(* Logix 5000 project; controller Thurs_Lab2 vendor 1 type 14 code 156 rev 30.11; software revision 30.00; part 3 of 5 *)
(* tags used below, declared in another part *)
   Action_015 : SFC_ACTION;
   Action_016 : SFC_ACTION;
   Action_017 : SFC_ACTION;
   Action_018 : SFC_ACTION;
   Action_019 : SFC_ACTION;
   Action_020 : SFC_ACTION;
   Action_021 : SFC_ACTION;
   Action_022 : SFC_ACTION;
   Action_023 : SFC_ACTION;
   Action_024 : SFC_ACTION;
   Step_000 : SFC_STEP;
   Step_011 : SFC_STEP;
   Step_012 : SFC_STEP;
   Step_013 : SFC_STEP;
   Step_015 : SFC_STEP;
   Step_016 : SFC_STEP;
   Step_017 : SFC_STEP;
   Step_018 : SFC_STEP;
   Step_019 : SFC_STEP;
   Step_020 : SFC_STEP;
   Step_021 : SFC_STEP;
   Tran_000 : BOOL;
   AUTO : BOOL;
   BYPASS : BOOL;
   CONTINUE : BOOL;
   CYCLE_START : BOOL;
   CYCLE_STOP : BOOL;
   CYLINDERSTATUS : DINT;
   DEEP : COUNTER;
   DELAY_PE_INPUT_PSB : TIMER;
   DRILL2 : DRILL2;
   ESTOP_PRESSED : BOOL;
   EXTEND : TIMER;
   FAULT : BOOL;
   LOAD_ONE_SHOT_SCAN : BOOL;
   M_PL0 : BOOL;
   M_PL1 : BOOL;
   M_PL2 : BOOL;
   M_PL3 : BOOL;
   M_PL4 : BOOL;
   M_PL5 : BOOL;
   M_WHEEL_MOTOR : BOOL;
   Man_ONE_SHOT_SCAN : BOOL;
   Manual : BOOL;
   MARK_CYL1 : CYLINDER;
   MARK_ONE_SHOT_SCAN : BOOL;
   MASTER_RESET_COUNT1 : COUNTER;
   MASTER_RESET_COUNT2 : COUNTER;
   MASTER_RESET_COUNT3 : COUNTER;
   MASTER_RESET_COUNT4 : COUNTER;
   MASTER_RESET_COUNT5 : COUNTER;
   MASTER_RESET_COUNT6 : COUNTER;
   MASTER_RESET_COUNT7 : COUNTER;
   ONE_SHOT_PSB0 : BOOL;
   ONE_SHOT_PSB1 : BOOL;
   OP1_STOP : BOOL;
   OP2_ONE_SHOT_SCAN : BOOL;
   OP2_STEP : DINT;
   OP2_STOP : BOOL;
   OP3_ONE_SHOT_SCAN : BOOL;
   OP3_STOP : BOOL;
   OP4_ONE_SHOT_SCAN : BOOL;
   OP4_STOP : BOOL;
   OP5_STOP : BOOL;
   OP6_MARK : TIMER;
   OP6_STOP : BOOL;
   OP7_STOP : BOOL;
   OPERATION : DINT;
   OPERATION_DONE : DINT;
   OPERATION_OFF : DINT;
   OUTPUT : INT;
   PAUSE : BOOL;
   PB0 : BOOL;
   PB1 : BOOL;
   PB2 : BOOL;
   PB3 : BOOL;
   PB4 : BOOL;
   PB5 : BOOL;
   PV_CYL1_EXT_SIG : BOOL;
   PV_CYL1_RET_SIG : BOOL;
   PV_CYL2_EXT_SIG : BOOL;
   PV_FAULT_RESET : BOOL;
   PV_MAX_DEPTH : DINT;
   PV_MIN_DEPTH : DINT;
   PV_MOTOR_START : BOOL;
   PV_RESET : BOOL;
   RESET : BOOL;
   SAFETY_RELAY_OFF : BOOL;
   SEQ_EN : BOOL;
   SHALLOW : COUNTER;
   SORT_ONE_SHOT_SCAN : BOOL;
   START_SIGNAL : BOOL;
   STATE : DINT;
   STEP : DINT;
   TEST_ONE_SHOT_SCAN : BOOL;
   Timer : TIMER;
   TOO_DEEP : BOOL;
   TOO_SHALLOW : BOOL;
(* MainProgram, continued *)

ROUTINE MainRoutine   (* ladder *)
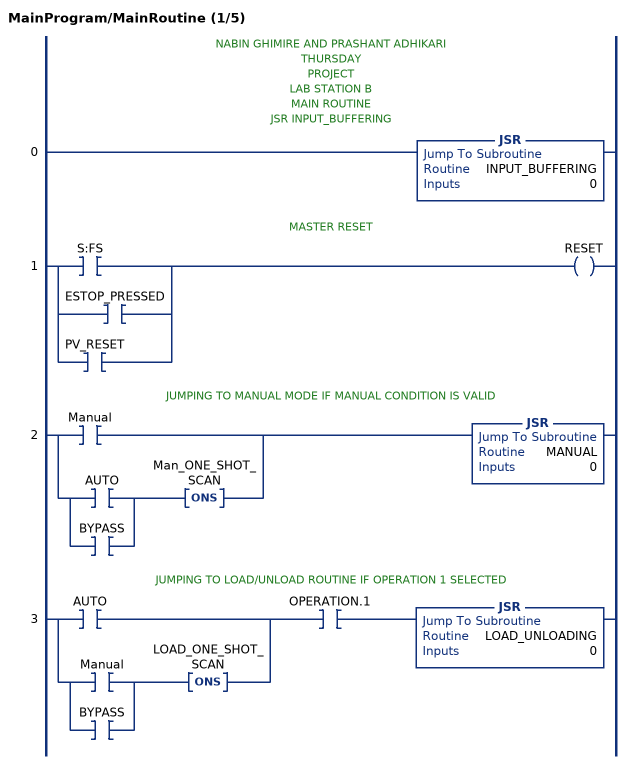
   // NABIN GHIMIRE AND PRASHANT ADHIKARI
   // THURSDAY
   // PROJECT
   // LAB STATION B
   // MAIN ROUTINE
   // JSR INPUT_BUFFERING
   0: JSR(INPUT_BUFFERING,0);
   // MASTER RESET
   1: [XIC(S:FS) ,XIC(ESTOP_PRESSED) ,XIC(PV_RESET) ]OTE(RESET);
   // JUMPING TO MANUAL MODE IF MANUAL CONDITION IS VALID
   2: [XIC(Manual) ,[XIC(AUTO) ,XIC(BYPASS) ] ONS(Man_ONE_SHOT_SCAN) ]JSR(MANUAL,0);
   // JUMPING TO LOAD/UNLOAD ROUTINE IF OPERATION 1 SELECTED
   3: [XIC(AUTO) ,[XIC(Manual) ,XIC(BYPASS) ] ONS(LOAD_ONE_SHOT_SCAN) ]XIC(OPERATION.1)JSR(LOAD_UNLOADING,0);
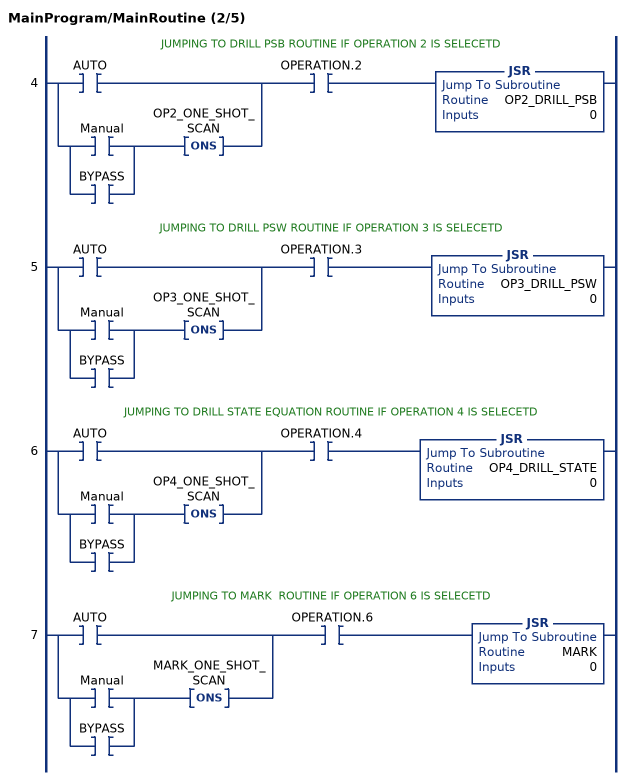
   // JUMPING TO DRILL PSB ROUTINE IF OPERATION 2 IS SELECETD
   4: [XIC(AUTO) ,[XIC(Manual) ,XIC(BYPASS) ] ONS(OP2_ONE_SHOT_SCAN) ]XIC(OPERATION.2)JSR(OP2_DRILL_PSB,0);
   // JUMPING TO DRILL PSW ROUTINE IF OPERATION 3 IS SELECETD
   5: [XIC(AUTO) ,[XIC(Manual) ,XIC(BYPASS) ] ONS(OP3_ONE_SHOT_SCAN) ]XIC(OPERATION.3)JSR(OP3_DRILL_PSW,0);
   // JUMPING TO DRILL STATE EQUATION ROUTINE IF OPERATION 4 IS SELECETD
   6: [XIC(AUTO) ,[XIC(Manual) ,XIC(BYPASS) ] ONS(OP4_ONE_SHOT_SCAN) ]XIC(OPERATION.4)JSR(OP4_DRILL_STATE,0);
   // JUMPING TO MARK  ROUTINE IF OPERATION 6 IS SELECETD
   7: [XIC(AUTO) ,[XIC(Manual) ,XIC(BYPASS) ] ONS(MARK_ONE_SHOT_SCAN) ]XIC(OPERATION.6)JSR(MARK,0);
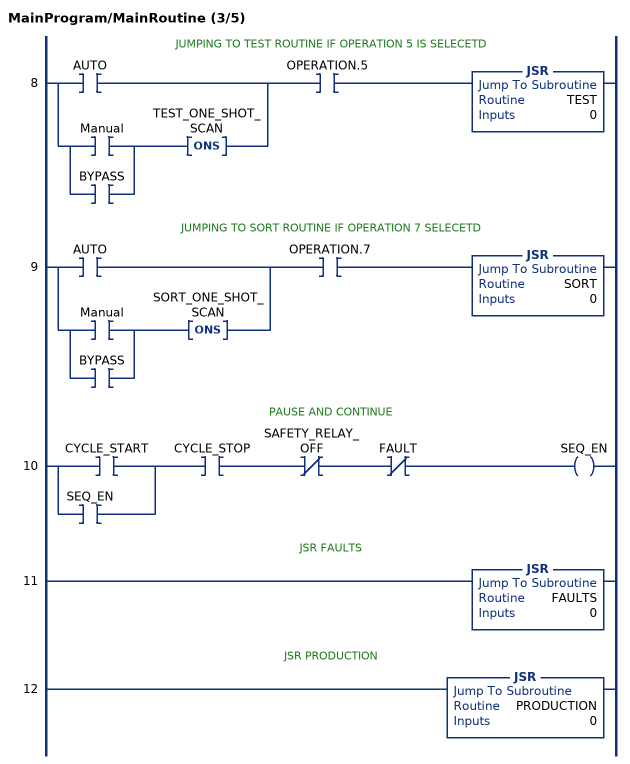
   // JUMPING TO TEST ROUTINE IF OPERATION 5 IS SELECETD
   8: [XIC(AUTO) ,[XIC(Manual) ,XIC(BYPASS) ] ONS(TEST_ONE_SHOT_SCAN) ]XIC(OPERATION.5)JSR(TEST,0);
   // JUMPING TO SORT ROUTINE IF OPERATION 7 SELECETD
   9: [XIC(AUTO) ,[XIC(Manual) ,XIC(BYPASS) ] ONS(SORT_ONE_SHOT_SCAN) ]XIC(OPERATION.7)JSR(SORT,0);
   // PAUSE AND CONTINUE
   10: [XIC(CYCLE_START) ,XIC(SEQ_EN) ]XIC(CYCLE_STOP)XIO(SAFETY_RELAY_OFF)XIO(FAULT)OTE(SEQ_EN);
   // JSR FAULTS
   11: JSR(FAULTS,0);
   // JSR PRODUCTION
   12: JSR(PRODUCTION,0);
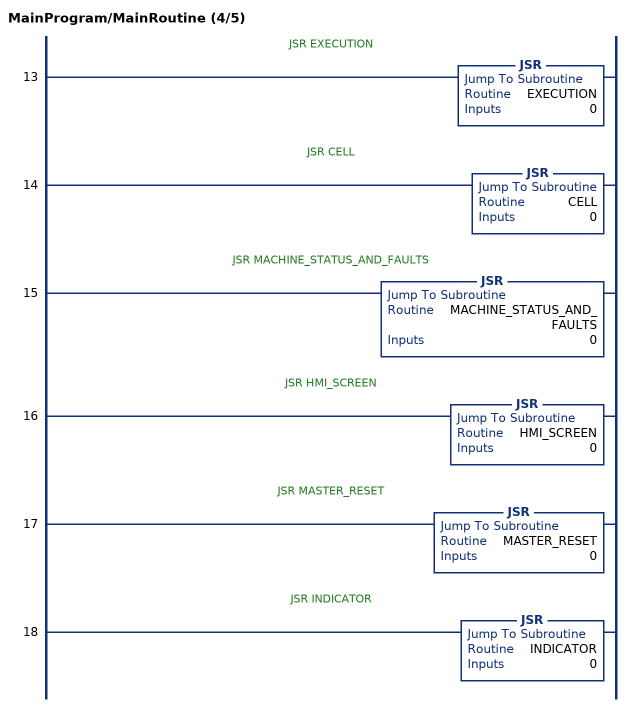
   // JSR EXECUTION
   13: JSR(EXECUTION,0);
   // JSR CELL
   14: JSR(CELL,0);
   // JSR MACHINE_STATUS_AND_FAULTS
   15: JSR(MACHINE_STATUS_AND_FAULTS,0);
   // JSR HMI_SCREEN
   16: JSR(HMI_SCREEN,0);
   // JSR MASTER_RESET
   17: JSR(MASTER_RESET,0);
   // JSR INDICATOR
   18: JSR(INDICATOR,0);
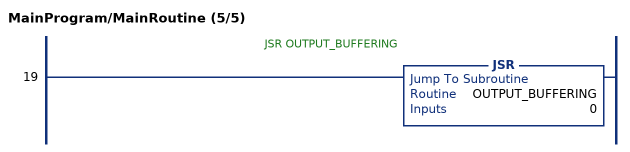
   // JSR OUTPUT_BUFFERING
   19: JSR(OUTPUT_BUFFERING,0);
END_ROUTINE

ROUTINE MANUAL   (* sequential function chart *)
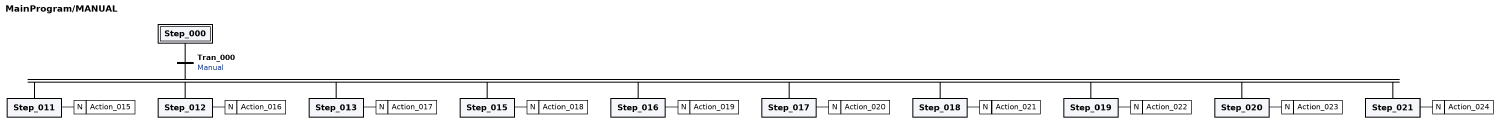
   // MANUAL ROUTINE USING SEQUENTIAL
   // FUNCTION CHART
   INITIAL_STEP Step_000:
   END_STEP
   TRANSITION Tran_000 FROM Step_000 TO (Step_012, Step_011, Step_013, Step_015, Step_016, Step_017, Step_018, Step_019, Step_020, Step_021)
      := Manual
         
         
   END_TRANSITION
   STEP Step_011:
      ACTION Action_015 (N):
         IF PB0 THEN
         	M_PL0:=1;
         ELSE
         	M_PL0:=0;
         END_IF;
         
         
      END_ACTION
   END_STEP
   STEP Step_012:
      ACTION Action_016 (N):
         IF PB1 THEN
         	M_PL1:=1;
         ELSE
         	M_PL1:=0;
         END_IF;
         
      END_ACTION
   END_STEP
   STEP Step_013:
      ACTION Action_017 (N):
         IF PB2 THEN
         	M_PL2:=1;
         ELSE
         	M_PL2:=0;
         END_IF;
         
      END_ACTION
   END_STEP
   STEP Step_015:
      ACTION Action_018 (N):
         IF PB3 THEN
         	M_PL3:=1;
         ELSE
         	M_PL3:=0;
         END_IF;
         
      END_ACTION
   END_STEP
   STEP Step_016:
      ACTION Action_019 (N):
         IF PB4 THEN
         	M_PL4:=1;
         ELSE
         	M_PL4:=0;
         END_IF;
         
      END_ACTION
   END_STEP
   STEP Step_017:
      ACTION Action_020 (N):
         IF PB5 THEN
         	M_PL5:=1;
         ELSE
         	M_PL5:=0;
         END_IF;
         
      END_ACTION
   END_STEP
   STEP Step_018:
      ACTION Action_021 (N):
         IF PV_MOTOR_START THEN
         	M_WHEEL_MOTOR:=1;
         ELSE
         	M_WHEEL_MOTOR:=0;
         END_IF;
         
      END_ACTION
   END_STEP
   STEP Step_019:
      ACTION Action_022 (N):
         IF PV_CYL2_EXT_SIG THEN
         	DRILL2.CYL2.EXT_SIG:=1;
         ELSE
         	DRILL2.CYL2.EXT_SIG:=0;
         END_IF;
         
      END_ACTION
   END_STEP
   STEP Step_020:
      ACTION Action_023 (N):
         IF PV_CYL1_RET_SIG THEN
         	DRILL2.CYL1.MAN_RET_SIG:=1;
         ELSE
         	DRILL2.CYL1.MAN_RET_SIG:=0;
         END_IF;
         
      END_ACTION
   END_STEP
   STEP Step_021:
      ACTION Action_024 (N):
         IF PV_CYL1_EXT_SIG THEN
         	DRILL2.CYL1.MAN_EXT_SIG:=1;
         ELSE
         	DRILL2.CYL1.MAN_EXT_SIG:=0;
         END_IF;
         
      END_ACTION
   END_STEP
END_ROUTINE

ROUTINE MARK   (* ladder *)
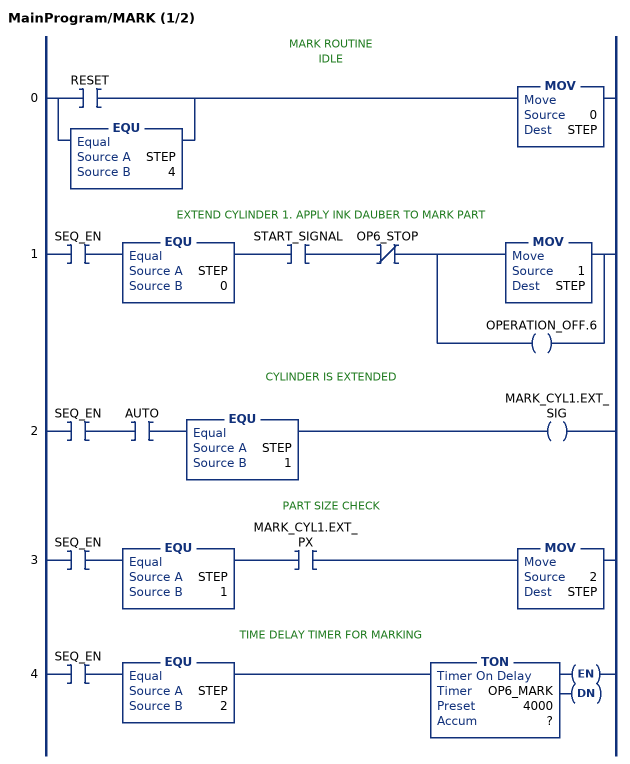
   // MARK ROUTINE
   // IDLE
   0: [XIC(RESET) ,EQU(STEP,4) ]MOV(0,STEP);
   // EXTEND CYLINDER 1. APPLY INK DAUBER TO MARK PART
   1: XIC(SEQ_EN)EQU(STEP,0)XIC(START_SIGNAL)XIO(OP6_STOP)[MOV(1,STEP) ,OTE(OPERATION_OFF.6) ];
   // CYLINDER IS EXTENDED
   2: XIC(SEQ_EN)XIC(AUTO)EQU(STEP,1)OTE(MARK_CYL1.EXT_SIG);
   // PART SIZE CHECK
   3: XIC(SEQ_EN)EQU(STEP,1)XIC(MARK_CYL1.EXT_PX)MOV(2,STEP);
   // TIME DELAY TIMER FOR MARKING
   4: XIC(SEQ_EN)EQU(STEP,2)TON(OP6_MARK,?,?);
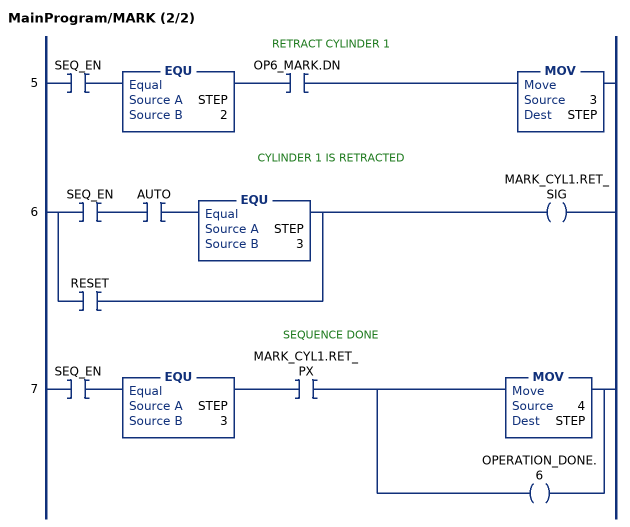
   // RETRACT CYLINDER 1
   5: XIC(SEQ_EN)EQU(STEP,2)XIC(OP6_MARK.DN)MOV(3,STEP);
   // CYLINDER 1 IS RETRACTED
   6: [XIC(SEQ_EN) XIC(AUTO) EQU(STEP,3) ,XIC(RESET) ]OTE(MARK_CYL1.RET_SIG);
   // SEQUENCE DONE
   7: XIC(SEQ_EN)EQU(STEP,3)XIC(MARK_CYL1.RET_PX)[MOV(4,STEP) ,OTE(OPERATION_DONE.6) ];
END_ROUTINE

ROUTINE MASTER_RESET   (* ladder *)
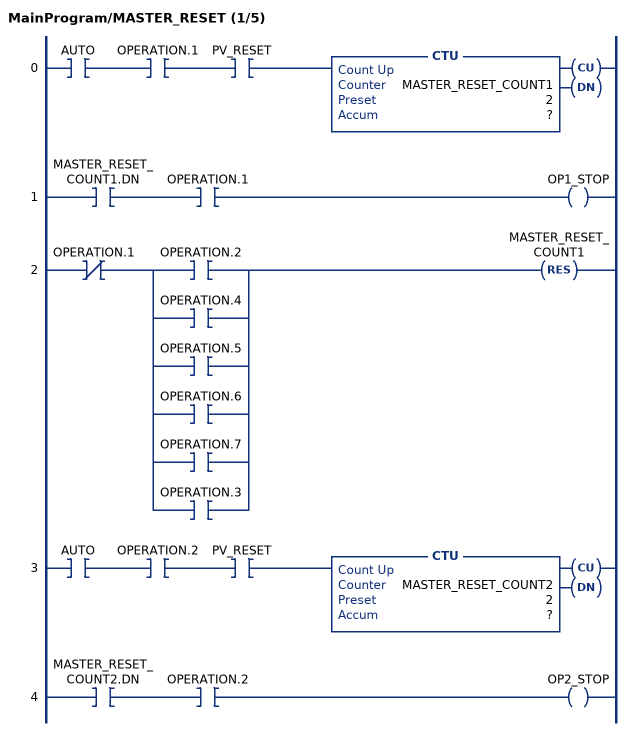
   0: XIC(AUTO)XIC(OPERATION.1)XIC(PV_RESET)CTU(MASTER_RESET_COUNT1,?,?);
   1: XIC(MASTER_RESET_COUNT1.DN)XIC(OPERATION.1)OTE(OP1_STOP);
   2: XIO(OPERATION.1)[XIC(OPERATION.2) ,XIC(OPERATION.4) ,XIC(OPERATION.5) ,XIC(OPERATION.6) ,XIC(OPERATION.7) ,XIC(OPERATION.3) ]RES(MASTER_RESET_COUNT1);
   3: XIC(AUTO)XIC(OPERATION.2)XIC(PV_RESET)CTU(MASTER_RESET_COUNT2,?,?);
   4: XIC(MASTER_RESET_COUNT2.DN)XIC(OPERATION.2)OTE(OP2_STOP);
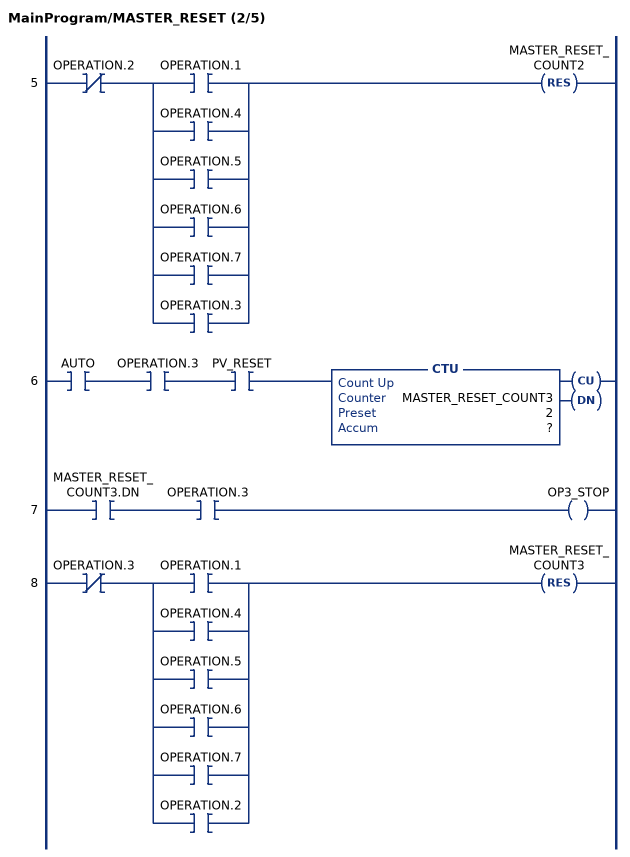
   5: XIO(OPERATION.2)[XIC(OPERATION.1) ,XIC(OPERATION.4) ,XIC(OPERATION.5) ,XIC(OPERATION.6) ,XIC(OPERATION.7) ,XIC(OPERATION.3) ]RES(MASTER_RESET_COUNT2);
   6: XIC(AUTO)XIC(OPERATION.3)XIC(PV_RESET)CTU(MASTER_RESET_COUNT3,?,?);
   7: XIC(MASTER_RESET_COUNT3.DN)XIC(OPERATION.3)OTE(OP3_STOP);
   8: XIO(OPERATION.3)[XIC(OPERATION.1) ,XIC(OPERATION.4) ,XIC(OPERATION.5) ,XIC(OPERATION.6) ,XIC(OPERATION.7) ,XIC(OPERATION.2) ]RES(MASTER_RESET_COUNT3);
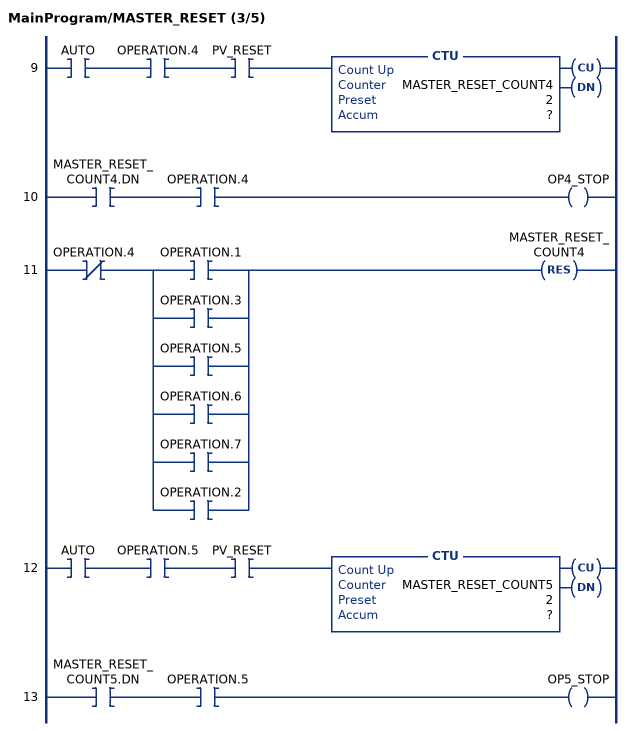
   9: XIC(AUTO)XIC(OPERATION.4)XIC(PV_RESET)CTU(MASTER_RESET_COUNT4,?,?);
   10: XIC(MASTER_RESET_COUNT4.DN)XIC(OPERATION.4)OTE(OP4_STOP);
   11: XIO(OPERATION.4)[XIC(OPERATION.1) ,XIC(OPERATION.3) ,XIC(OPERATION.5) ,XIC(OPERATION.6) ,XIC(OPERATION.7) ,XIC(OPERATION.2) ]RES(MASTER_RESET_COUNT4);
   12: XIC(AUTO)XIC(OPERATION.5)XIC(PV_RESET)CTU(MASTER_RESET_COUNT5,?,?);
   13: XIC(MASTER_RESET_COUNT5.DN)XIC(OPERATION.5)OTE(OP5_STOP);
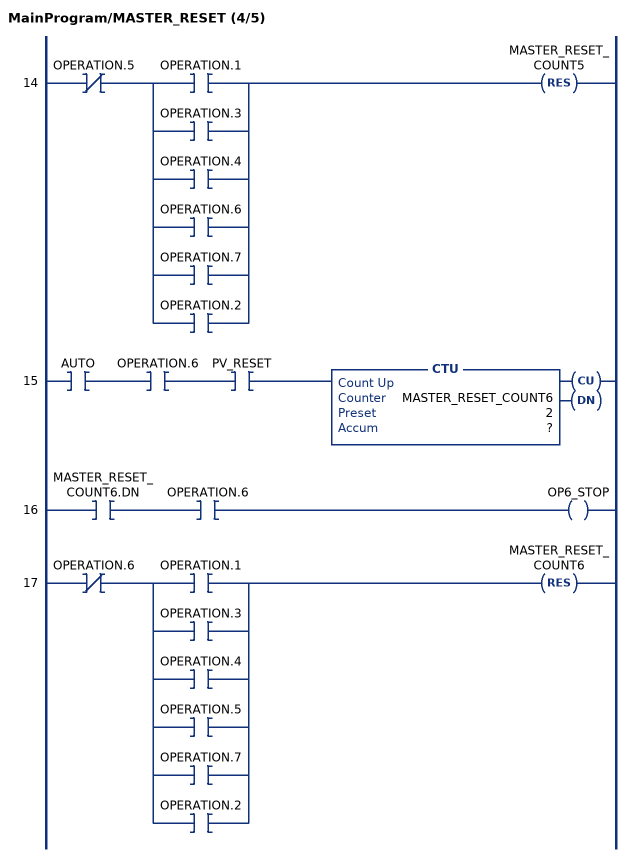
   14: XIO(OPERATION.5)[XIC(OPERATION.1) ,XIC(OPERATION.3) ,XIC(OPERATION.4) ,XIC(OPERATION.6) ,XIC(OPERATION.7) ,XIC(OPERATION.2) ]RES(MASTER_RESET_COUNT5);
   15: XIC(AUTO)XIC(OPERATION.6)XIC(PV_RESET)CTU(MASTER_RESET_COUNT6,?,?);
   16: XIC(MASTER_RESET_COUNT6.DN)XIC(OPERATION.6)OTE(OP6_STOP);
   17: XIO(OPERATION.6)[XIC(OPERATION.1) ,XIC(OPERATION.3) ,XIC(OPERATION.4) ,XIC(OPERATION.5) ,XIC(OPERATION.7) ,XIC(OPERATION.2) ]RES(MASTER_RESET_COUNT6);
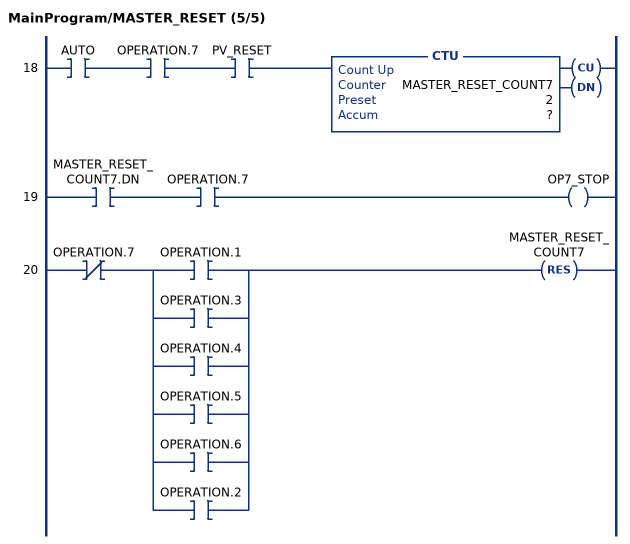
   18: XIC(AUTO)XIC(OPERATION.7)XIC(PV_RESET)CTU(MASTER_RESET_COUNT7,?,?);
   19: XIC(MASTER_RESET_COUNT7.DN)XIC(OPERATION.7)OTE(OP7_STOP);
   20: XIO(OPERATION.7)[XIC(OPERATION.1) ,XIC(OPERATION.3) ,XIC(OPERATION.4) ,XIC(OPERATION.5) ,XIC(OPERATION.6) ,XIC(OPERATION.2) ]RES(MASTER_RESET_COUNT7);
END_ROUTINE

ROUTINE OP2_DRILL_PSB   (* ladder *)
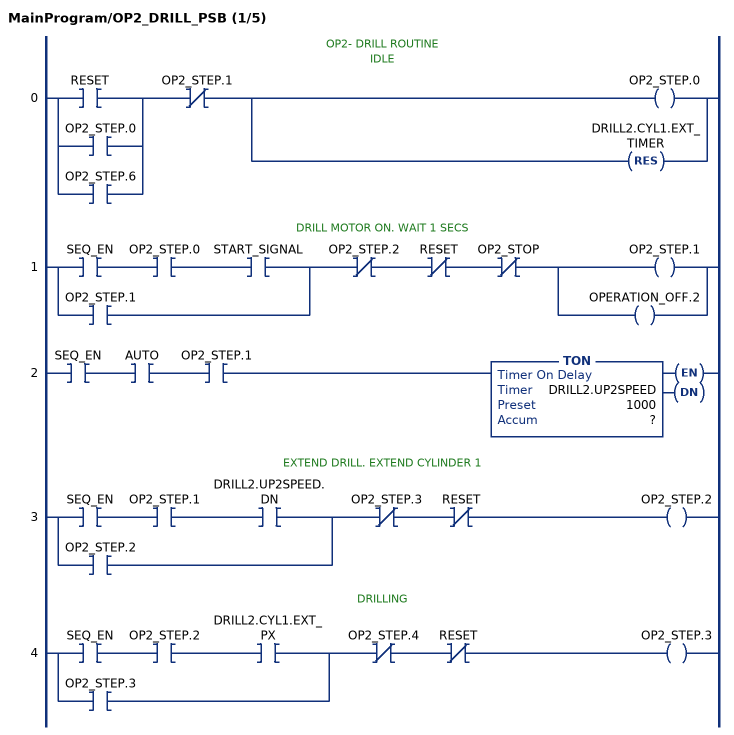
   // OP2- DRILL ROUTINE
   // IDLE
   0: [XIC(RESET) ,XIC(OP2_STEP.0) ,XIC(OP2_STEP.6) ]XIO(OP2_STEP.1)[OTE(OP2_STEP.0) ,RES(DRILL2.CYL1.EXT_TIMER) ];
   // DRILL MOTOR ON. WAIT 1 SECS
   1: [XIC(SEQ_EN) XIC(OP2_STEP.0) XIC(START_SIGNAL) ,XIC(OP2_STEP.1) ]XIO(OP2_STEP.2)XIO(RESET)XIO(OP2_STOP)[OTE(OP2_STEP.1) ,OTE(OPERATION_OFF.2) ];
   2: XIC(SEQ_EN)XIC(AUTO)XIC(OP2_STEP.1)TON(DRILL2.UP2SPEED,?,?);
   // EXTEND DRILL. EXTEND CYLINDER 1
   3: [XIC(SEQ_EN) XIC(OP2_STEP.1) XIC(DRILL2.UP2SPEED.DN) ,XIC(OP2_STEP.2) ]XIO(OP2_STEP.3)XIO(RESET)OTE(OP2_STEP.2);
   // DRILLING
   4: [XIC(SEQ_EN) XIC(OP2_STEP.2) XIC(DRILL2.CYL1.EXT_PX) ,XIC(OP2_STEP.3) ]XIO(OP2_STEP.4)XIO(RESET)OTE(OP2_STEP.3);
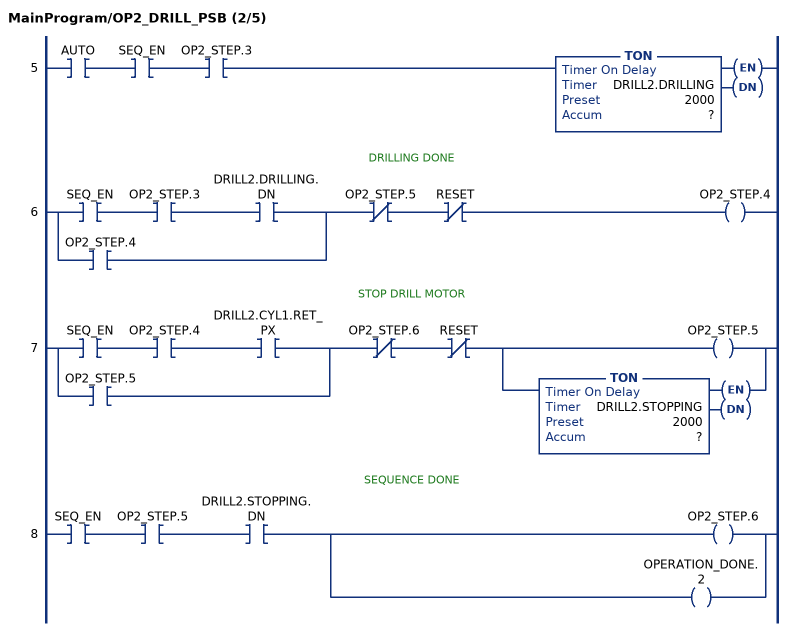
   5: XIC(AUTO)XIC(SEQ_EN)XIC(OP2_STEP.3)TON(DRILL2.DRILLING,?,?);
   // DRILLING DONE
   6: [XIC(SEQ_EN) XIC(OP2_STEP.3) XIC(DRILL2.DRILLING.DN) ,XIC(OP2_STEP.4) ]XIO(OP2_STEP.5)XIO(RESET)OTE(OP2_STEP.4);
   // STOP DRILL MOTOR
   7: [XIC(SEQ_EN) XIC(OP2_STEP.4) XIC(DRILL2.CYL1.RET_PX) ,XIC(OP2_STEP.5) ]XIO(OP2_STEP.6)XIO(RESET)[OTE(OP2_STEP.5) ,TON(DRILL2.STOPPING,?,?) ];
   // SEQUENCE DONE
   8: XIC(SEQ_EN)XIC(OP2_STEP.5)XIC(DRILL2.STOPPING.DN)[OTE(OP2_STEP.6) ,OTE(OPERATION_DONE.2) ];
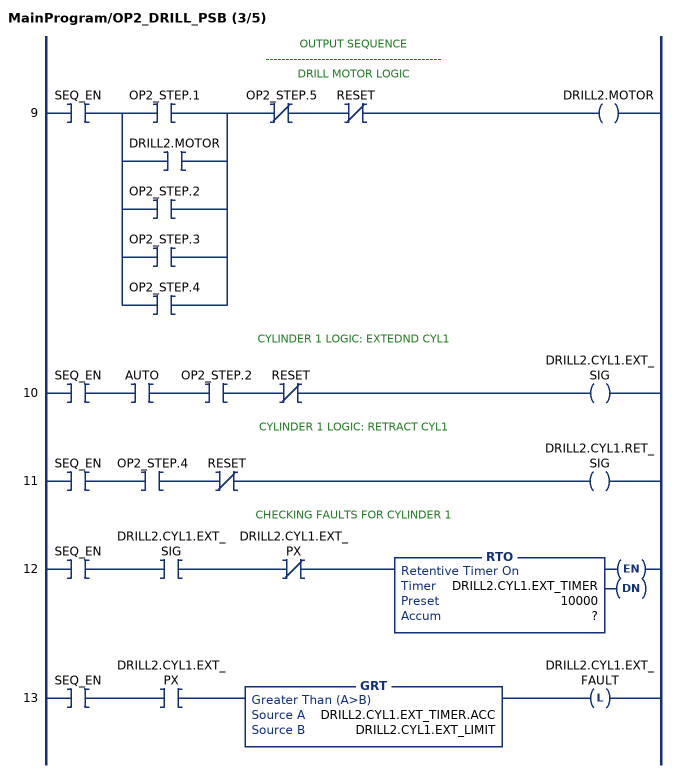
   // OUTPUT SEQUENCE
   // --------------------------------------------
   // DRILL MOTOR LOGIC
   9: XIC(SEQ_EN)[XIC(OP2_STEP.1) ,XIC(DRILL2.MOTOR) ,XIC(OP2_STEP.2) ,XIC(OP2_STEP.3) ,XIC(OP2_STEP.4) ]XIO(OP2_STEP.5)XIO(RESET)OTE(DRILL2.MOTOR);
   // CYLINDER 1 LOGIC: EXTEDND CYL1
   10: XIC(SEQ_EN)XIC(AUTO)XIC(OP2_STEP.2)XIO(RESET)OTE(DRILL2.CYL1.EXT_SIG);
   // CYLINDER 1 LOGIC: RETRACT CYL1
   11: XIC(SEQ_EN)XIC(OP2_STEP.4)XIO(RESET)OTE(DRILL2.CYL1.RET_SIG);
   // CHECKING FAULTS FOR CYLINDER 1
   12: XIC(SEQ_EN)XIC(DRILL2.CYL1.EXT_SIG)XIO(DRILL2.CYL1.EXT_PX)RTO(DRILL2.CYL1.EXT_TIMER,?,?);
   13: XIC(SEQ_EN)XIC(DRILL2.CYL1.EXT_PX)GRT(DRILL2.CYL1.EXT_TIMER.ACC,DRILL2.CYL1.EXT_LIMIT)OTL(DRILL2.CYL1.EXT_FAULT);
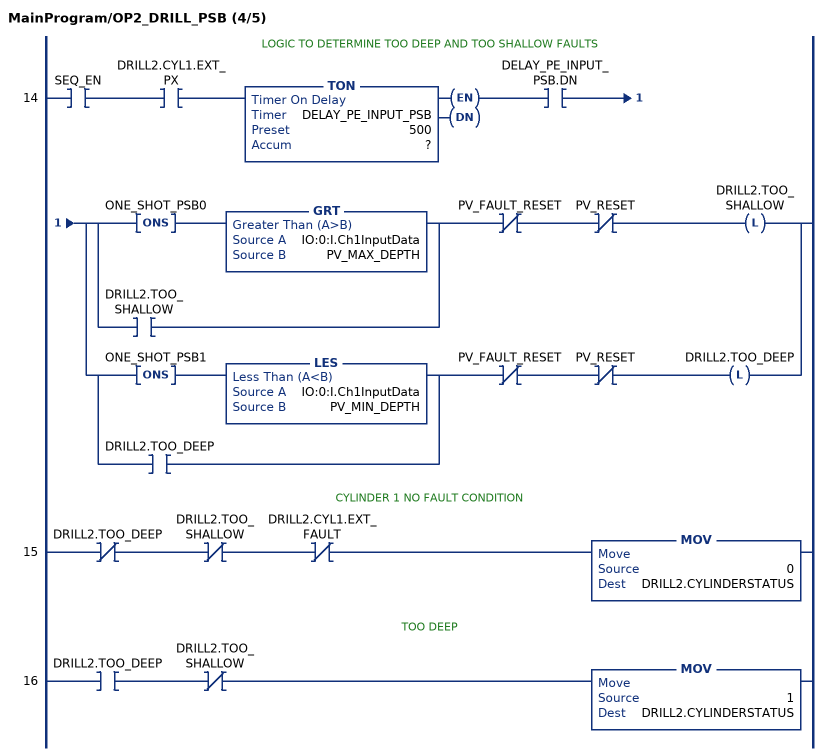
   // LOGIC TO DETERMINE TOO DEEP AND TOO SHALLOW FAULTS
   14: XIC(SEQ_EN)XIC(DRILL2.CYL1.EXT_PX)TON(DELAY_PE_INPUT_PSB,?,?)XIC(DELAY_PE_INPUT_PSB.DN)[[ONS(ONE_SHOT_PSB0) GRT(IO:0:I.Ch1InputData,PV_MAX_DEPTH) ,XIC(DRILL2.TOO_SHALLOW) ] XIO(PV_FAULT_RESET) XIO(PV_RESET) OTL(DRILL2.TOO_SHALLOW) ,[ONS(ONE_SHOT_PSB1) LES(IO:0:I.Ch1InputData,PV_MIN_DEPTH) ,XIC(DRILL2.TOO_DEEP) ] XIO(PV_FAULT_RESET) XIO(PV_RESET) OTL(DRILL2.TOO_DEEP) ];
   // CYLINDER 1 NO FAULT CONDITION
   15: XIO(DRILL2.TOO_DEEP)XIO(DRILL2.TOO_SHALLOW)XIO(DRILL2.CYL1.EXT_FAULT)MOV(0,DRILL2.CYLINDERSTATUS);
   // TOO DEEP
   16: XIC(DRILL2.TOO_DEEP)XIO(DRILL2.TOO_SHALLOW)MOV(1,DRILL2.CYLINDERSTATUS);
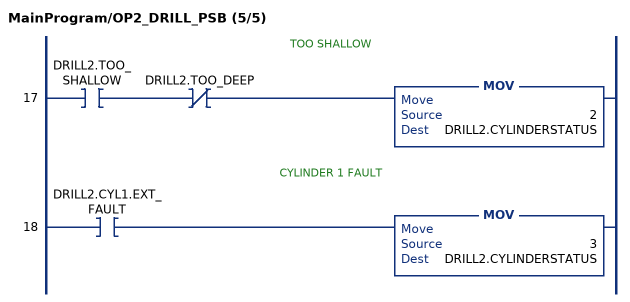
   // TOO SHALLOW
   17: XIC(DRILL2.TOO_SHALLOW)XIO(DRILL2.TOO_DEEP)MOV(2,DRILL2.CYLINDERSTATUS);
   // CYLINDER 1 FAULT
   18: XIC(DRILL2.CYL1.EXT_FAULT)MOV(3,DRILL2.CYLINDERSTATUS);
END_ROUTINE
